// SIMATIC S7-200 project (STEP 7-Micro/WIN), CPU 224XP CN REL 02.01

ORGANIZATION_BLOCK MAIN:OB1
TITLE= 
// PROGRAM COMMENTS
// Press F1 for help and example program
//  
BEGIN
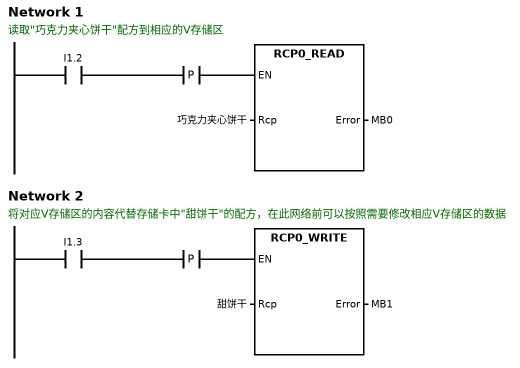
Network 1
// 读取"巧克力夹心饼干"配方到相应的V存储区
// (network saved uncompiled; LAD cells follow)
// row 0: c0 -| |- I1.2  c1 -|P|-  c2 [RCP0_READ EN:=power@row0, Rcp:=巧克力夹心饼干, Error=>MB0]
// row 1: c2 [box]
Network 2
// 将对应V存储区的内容代替存储卡中"甜饼干"的配方，在此网络前可以按照需要修改相应V存储区的数据
// (network saved uncompiled; LAD cells follow)
// row 0: c0 -| |- I1.3  c1 -|P|-  c2 [RCP0_WRITE EN:=power@row0, Rcp:=甜饼干, Error=>MB1]
// row 1: c2 [box]
END_ORGANIZATION_BLOCK

// SBR1: protected block, not included

// SBR2: protected block, not included

// (further data pages could not be read)
